INTERFACE I_JsonDeserializer EXTENDS I_Deserializer, I_EventEmitter, I_Disposable

END_INTERFACE

(* stored: Version 1.1.0.1, ProductVersion 3.1.4024.12
   Itf I_JsonDeserializer: Id {4a3f3e10-0467-485e-85cf-f526fb6a2a91} *)
